PROGRAM POU_2
VAR
END_VAR

END_PROGRAM

(* stored: Version 1.1.0.1, ProductVersion 3.1.4024.12
   POU POU_2: Id {5dd7250e-f1a5-4f25-b632-9e9acc7716d7}, SpecialFunc None *)
